TYPE STRING_5K : STRING(5000); END_TYPE

(* stored: Version 1.1.0.1, ProductVersion 3.1.4024.11
   DUT STRING_5K: Id {814ccfa5-194c-47af-86ae-d9b8b77e2b62} *)
